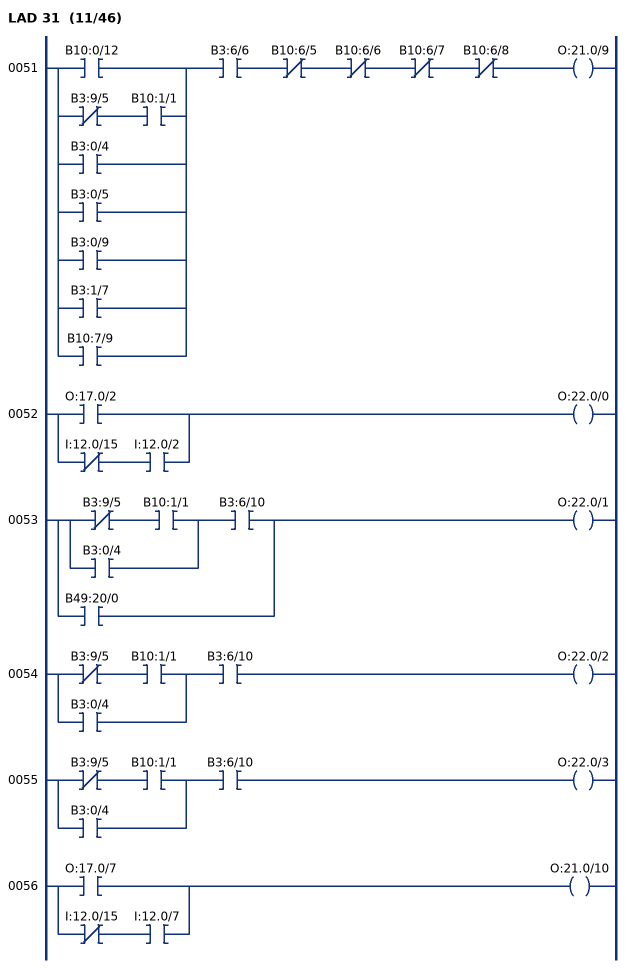
% Rung: 51 %
SOR BST XIC B10:0/12 NXB XIO B3:9/5 XIC B10:1/1 NXB XIC B3:0/4 NXB XIC B3:0/5 NXB XIC B3:0/9 NXB XIC B3:1/7 NXB XIC B10:7/9 BND XIC B3:6/6 XIO B10:6/5 XIO B10:6/6 XIO B10:6/7 XIO B10:6/8 OTE O:21.0/9 EOR
% Rung: 52 %
SOR BST XIC O:17.0/2 NXB XIO I:12.0/15 XIC I:12.0/2 BND OTE O:22.0/0 EOR
% Rung: 53 %
SOR BST BST XIO B3:9/5 XIC B10:1/1 NXB XIC B3:0/4 BND XIC B3:6/10 NXB XIC B49:20/0 BND OTE O:22.0/1 EOR
% Rung: 54 %
SOR BST XIO B3:9/5 XIC B10:1/1 NXB XIC B3:0/4 BND XIC B3:6/10 OTE O:22.0/2 EOR
% Rung: 55 %
SOR BST XIO B3:9/5 XIC B10:1/1 NXB XIC B3:0/4 BND XIC B3:6/10 OTE O:22.0/3 EOR
% Rung: 56 %
SOR BST XIC O:17.0/7 NXB XIO I:12.0/15 XIC I:12.0/7 BND OTE O:21.0/10 EOR

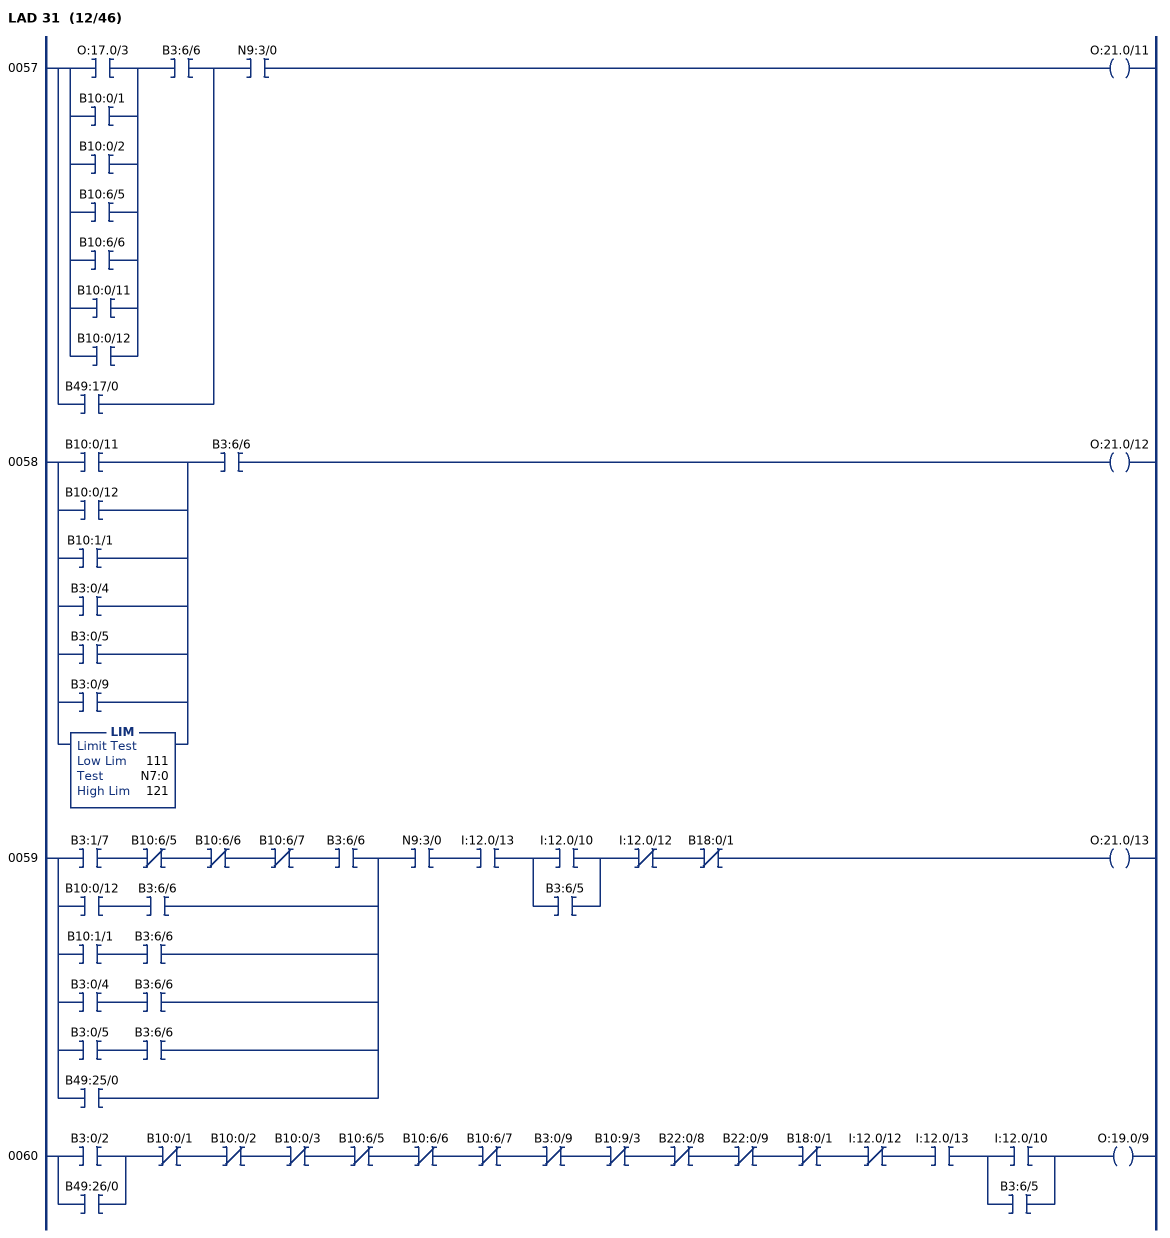
% Rung: 57 %
SOR BST BST XIC O:17.0/3 NXB XIC B10:0/1 NXB XIC B10:0/2 NXB XIC B10:6/5 NXB XIC B10:6/6 NXB XIC B10:0/11 NXB XIC B10:0/12 BND XIC B3:6/6 NXB XIC B49:17/0 BND XIC N9:3/0 OTE O:21.0/11 EOR
% Rung: 58 %
SOR BST XIC B10:0/11 NXB XIC B10:0/12 NXB XIC B10:1/1 NXB XIC B3:0/4 NXB XIC B3:0/5 NXB XIC B3:0/9 NXB LIM 111 N7:0 121 BND XIC B3:6/6 OTE O:21.0/12 EOR
% Rung: 59 %
SOR BST XIC B3:1/7 XIO B10:6/5 XIO B10:6/6 XIO B10:6/7 XIC B3:6/6 NXB XIC B10:0/12 XIC B3:6/6 NXB XIC B10:1/1 XIC B3:6/6 NXB XIC B3:0/4 XIC B3:6/6 NXB XIC B3:0/5 XIC B3:6/6 NXB XIC B49:25/0 BND XIC N9:3/0 XIC I:12.0/13 BST XIC I:12.0/10 NXB XIC B3:6/5 BND XIO I:12.0/12 XIO B18:0/1 OTE O:21.0/13 EOR
% Rung: 60 %
SOR BST XIC B3:0/2 NXB XIC B49:26/0 BND XIO B10:0/1 XIO B10:0/2 XIO B10:0/3 XIO B10:6/5 XIO B10:6/6 XIO B10:6/7 XIO B3:0/9 XIO B10:9/3 XIO B22:0/8 XIO B22:0/9 XIO B18:0/1 XIO I:12.0/12 XIC I:12.0/13 BST XIC I:12.0/10 NXB XIC B3:6/5 BND OTE O:19.0/9 EOR

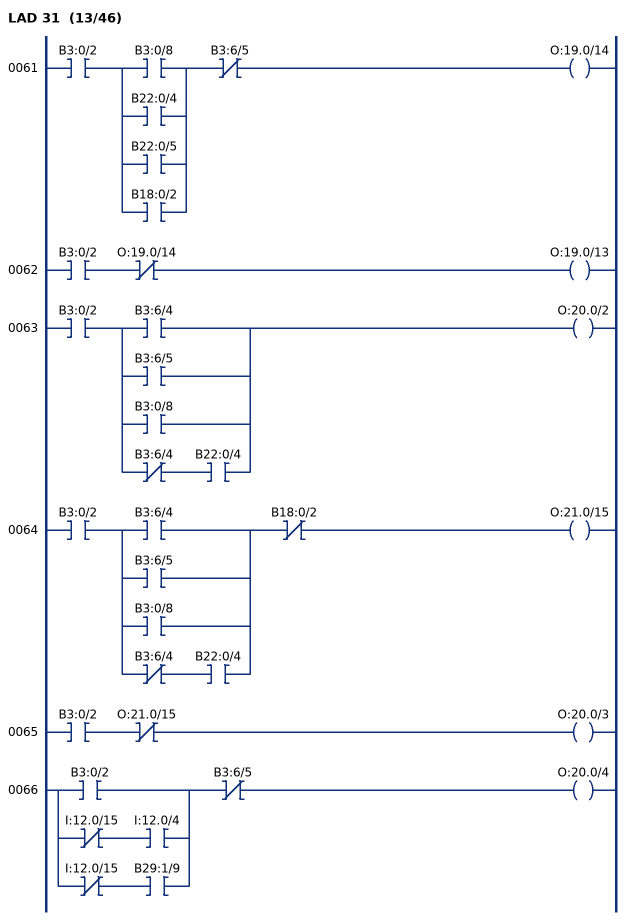
% Rung: 61 %
SOR XIC B3:0/2 BST XIC B3:0/8 NXB XIC B22:0/4 NXB XIC B22:0/5 NXB XIC B18:0/2 BND XIO B3:6/5 OTE O:19.0/14 EOR
% Rung: 62 %
SOR XIC B3:0/2 XIO O:19.0/14 OTE O:19.0/13 EOR
% Rung: 63 %
SOR XIC B3:0/2 BST XIC B3:6/4 NXB XIC B3:6/5 NXB XIC B3:0/8 NXB XIO B3:6/4 XIC B22:0/4 BND OTE O:20.0/2 EOR
% Rung: 64 %
SOR XIC B3:0/2 BST XIC B3:6/4 NXB XIC B3:6/5 NXB XIC B3:0/8 NXB XIO B3:6/4 XIC B22:0/4 BND XIO B18:0/2 OTE O:21.0/15 EOR
% Rung: 65 %
SOR XIC B3:0/2 XIO O:21.0/15 OTE O:20.0/3 EOR
% Rung: 66 %
SOR BST XIC B3:0/2 NXB XIO I:12.0/15 XIC I:12.0/4 NXB XIO I:12.0/15 XIC B29:1/9 BND XIO B3:6/5 OTE O:20.0/4 EOR

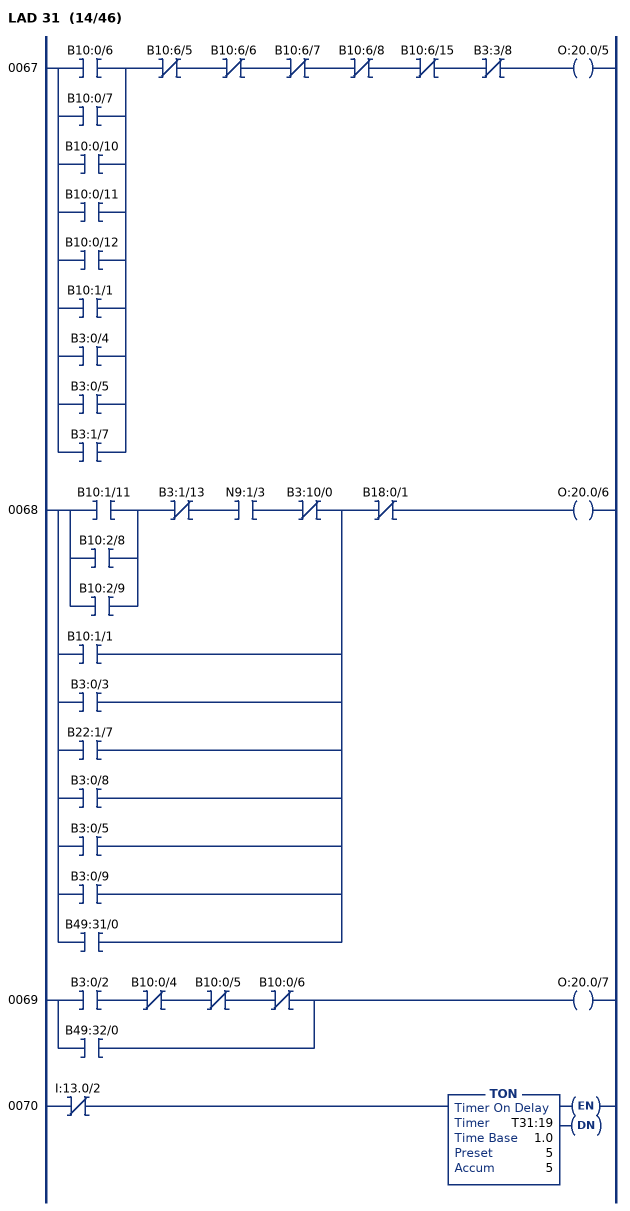
% Rung: 67 %
SOR BST XIC B10:0/6 NXB XIC B10:0/7 NXB XIC B10:0/10 NXB XIC B10:0/11 NXB XIC B10:0/12 NXB XIC B10:1/1 NXB XIC B3:0/4 NXB XIC B3:0/5 NXB XIC B3:1/7 BND XIO B10:6/5 XIO B10:6/6 XIO B10:6/7 XIO B10:6/8 XIO B10:6/15 XIO B3:3/8 OTE O:20.0/5 EOR
% Rung: 68 %
SOR BST BST XIC B10:1/11 NXB XIC B10:2/8 NXB XIC B10:2/9 BND XIO B3:1/13 XIC N9:1/3 XIO B3:10/0 NXB XIC B10:1/1 NXB XIC B3:0/3 NXB XIC B22:1/7 NXB XIC B3:0/8 NXB XIC B3:0/5 NXB XIC B3:0/9 NXB XIC B49:31/0 BND XIO B18:0/1 OTE O:20.0/6 EOR
% Rung: 69 %
SOR BST XIC B3:0/2 XIO B10:0/4 XIO B10:0/5 XIO B10:0/6 NXB XIC B49:32/0 BND OTE O:20.0/7 EOR
% Rung: 70 %
SOR XIO I:13.0/2 TON T31:19 1.0 5 5 EOR

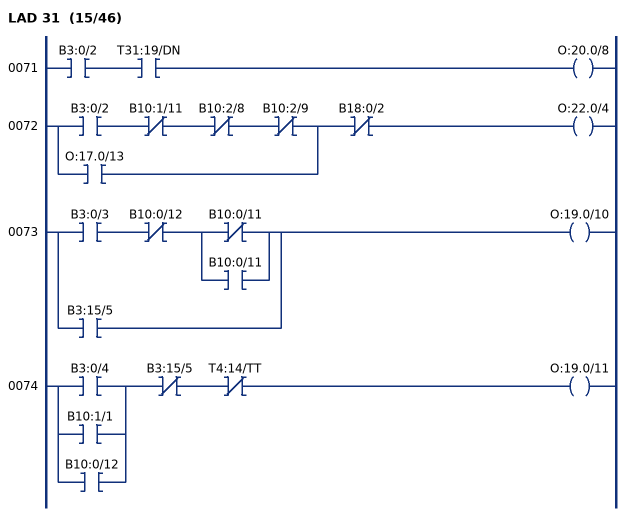
% Rung: 71 %
SOR XIC B3:0/2 XIC T31:19/DN OTE O:20.0/8 EOR
% Rung: 72 %
SOR BST XIC B3:0/2 XIO B10:1/11 XIO B10:2/8 XIO B10:2/9 NXB XIC O:17.0/13 BND XIO B18:0/2 OTE O:22.0/4 EOR
% Rung: 73 %
SOR BST XIC B3:0/3 XIO B10:0/12 BST XIO B10:0/11 NXB XIC B10:0/11 BND NXB XIC B3:15/5 BND OTE O:19.0/10 EOR
% Rung: 74 %
SOR BST XIC B3:0/4 NXB XIC B10:1/1 NXB XIC B10:0/12 BND XIO B3:15/5 XIO T4:14/TT OTE O:19.0/11 EOR

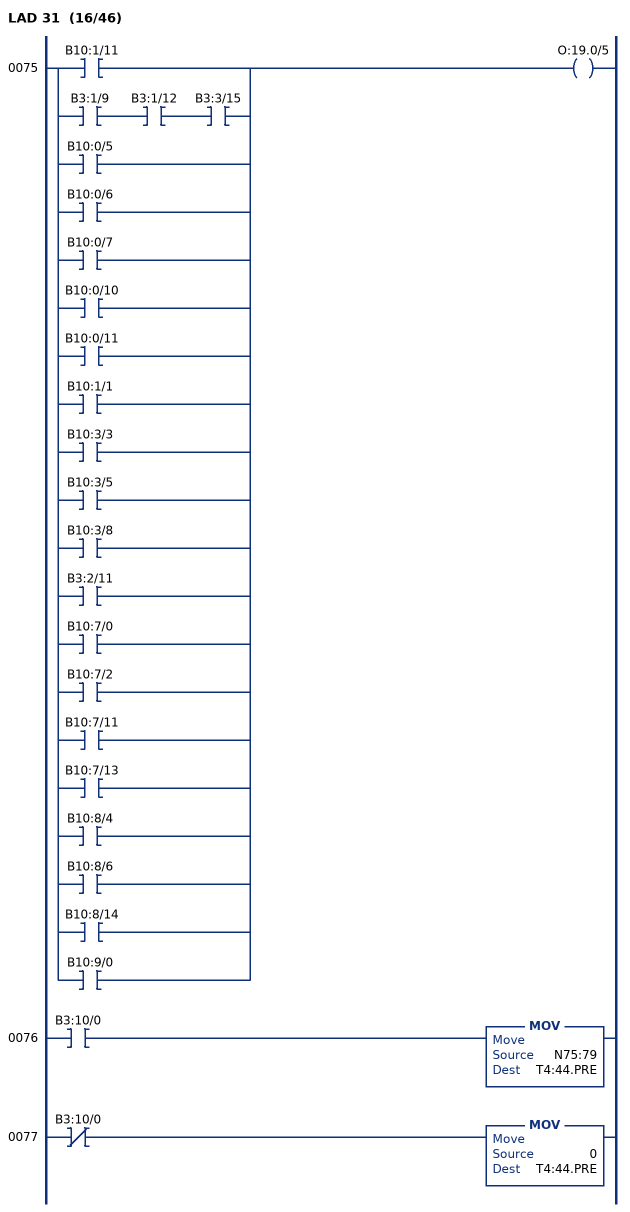
% Rung: 75 %
SOR BST XIC B10:1/11 NXB XIC B3:1/9 XIC B3:1/12 XIC B3:3/15 NXB XIC B10:0/5 NXB XIC B10:0/6 NXB XIC B10:0/7 NXB XIC B10:0/10 NXB XIC B10:0/11 NXB XIC B10:1/1 NXB XIC B10:3/3 NXB XIC B10:3/5 NXB XIC B10:3/8 NXB XIC B3:2/11 NXB XIC B10:7/0 NXB XIC B10:7/2 NXB XIC B10:7/11 NXB XIC B10:7/13 NXB XIC B10:8/4 NXB XIC B10:8/6 NXB XIC B10:8/14 NXB XIC B10:9/0 BND OTE O:19.0/5 EOR
% Rung: 76 %
SOR XIC B3:10/0 MOV N75:79 T4:44.PRE EOR
% Rung: 77 %
SOR XIO B3:10/0 MOV 0 T4:44.PRE EOR

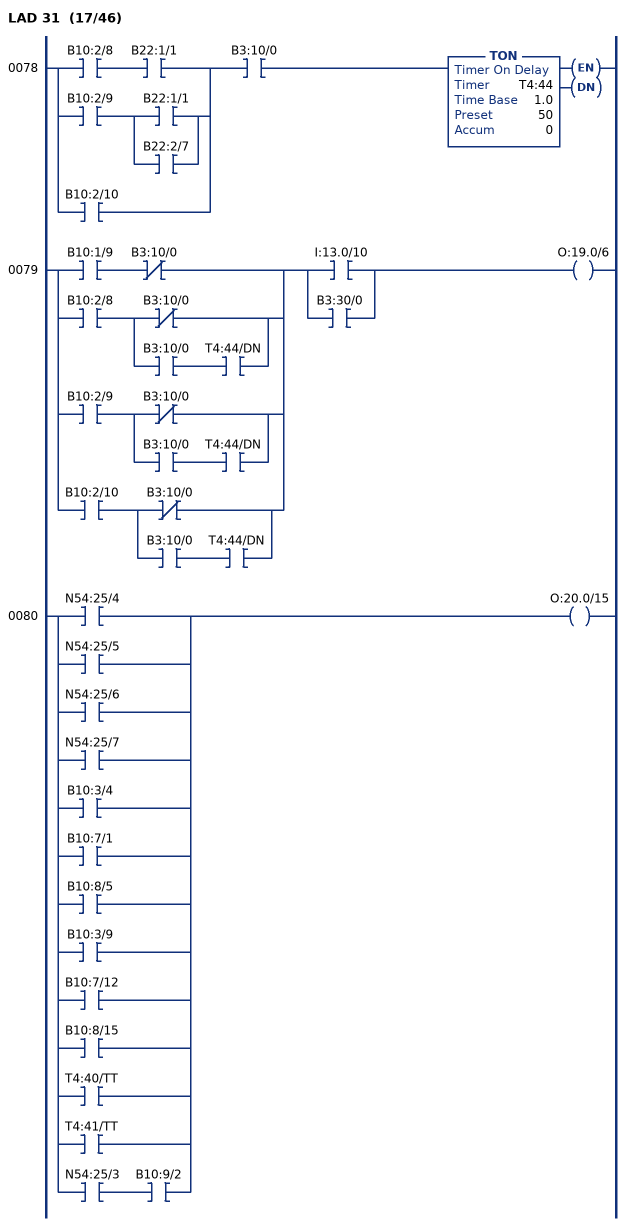
% Rung: 78 %
SOR BST XIC B10:2/8 XIC B22:1/1 NXB XIC B10:2/9 BST XIC B22:1/1 NXB XIC B22:2/7 BND NXB XIC B10:2/10 BND XIC B3:10/0 TON T4:44 1.0 50 0 EOR
% Rung: 79 %
SOR BST XIC B10:1/9 XIO B3:10/0 NXB XIC B10:2/8 BST XIO B3:10/0 NXB XIC B3:10/0 XIC T4:44/DN BND NXB XIC B10:2/9 BST XIO B3:10/0 NXB XIC B3:10/0 XIC T4:44/DN BND NXB XIC B10:2/10 BST XIO B3:10/0 NXB XIC B3:10/0 XIC T4:44/DN BND BND BST XIC I:13.0/10 NXB XIC B3:30/0 BND OTE O:19.0/6 EOR
% Rung: 80 %
SOR BST XIC N54:25/4 NXB XIC N54:25/5 NXB XIC N54:25/6 NXB XIC N54:25/7 NXB XIC B10:3/4 NXB XIC B10:7/1 NXB XIC B10:8/5 NXB XIC B10:3/9 NXB XIC B10:7/12 NXB XIC B10:8/15 NXB XIC T4:40/TT NXB XIC T4:41/TT NXB XIC N54:25/3 XIC B10:9/2 BND OTE O:20.0/15 EOR

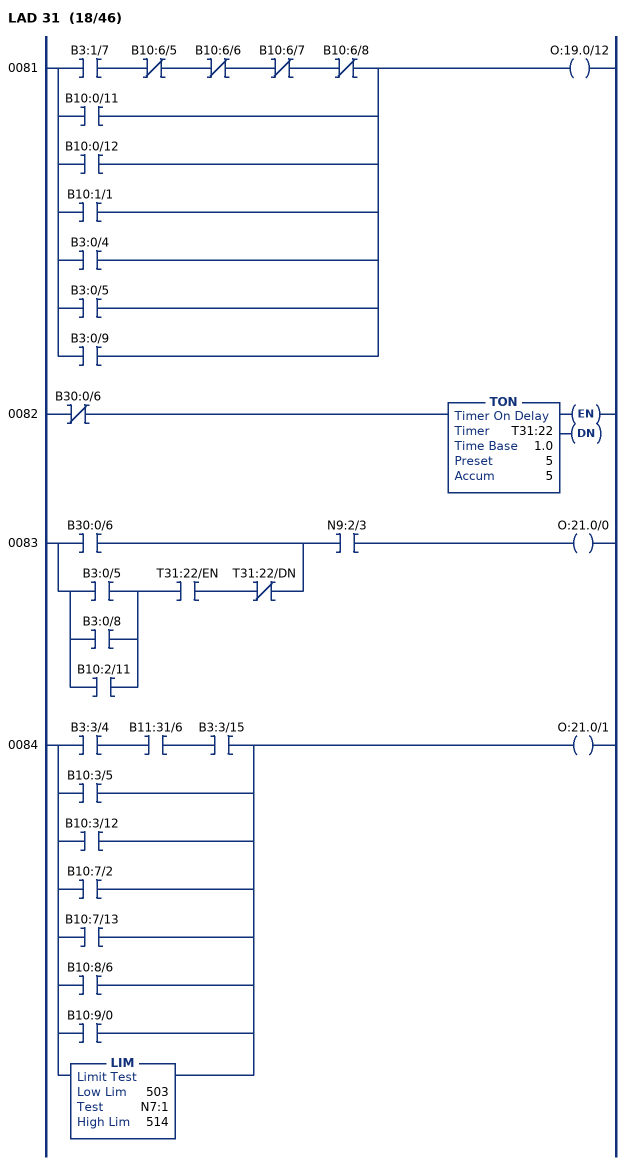
% Rung: 81 %
SOR BST XIC B3:1/7 XIO B10:6/5 XIO B10:6/6 XIO B10:6/7 XIO B10:6/8 NXB XIC B10:0/11 NXB XIC B10:0/12 NXB XIC B10:1/1 NXB XIC B3:0/4 NXB XIC B3:0/5 NXB XIC B3:0/9 BND OTE O:19.0/12 EOR
% Rung: 82 %
SOR XIO B30:0/6 TON T31:22 1.0 5 5 EOR
% Rung: 83 %
SOR BST XIC B30:0/6 NXB BST XIC B3:0/5 NXB XIC B3:0/8 NXB XIC B10:2/11 BND XIC T31:22/EN XIO T31:22/DN BND XIC N9:2/3 OTE O:21.0/0 EOR
% Rung: 84 %
SOR BST XIC B3:3/4 XIC B11:31/6 XIC B3:3/15 NXB BST XIC B10:3/5 NXB XIC B10:3/12 NXB XIC B10:7/2 NXB XIC B10:7/13 NXB XIC B10:8/6 NXB XIC B10:9/0 NXB LIM 503 N7:1 514 BND BND OTE O:21.0/1 EOR

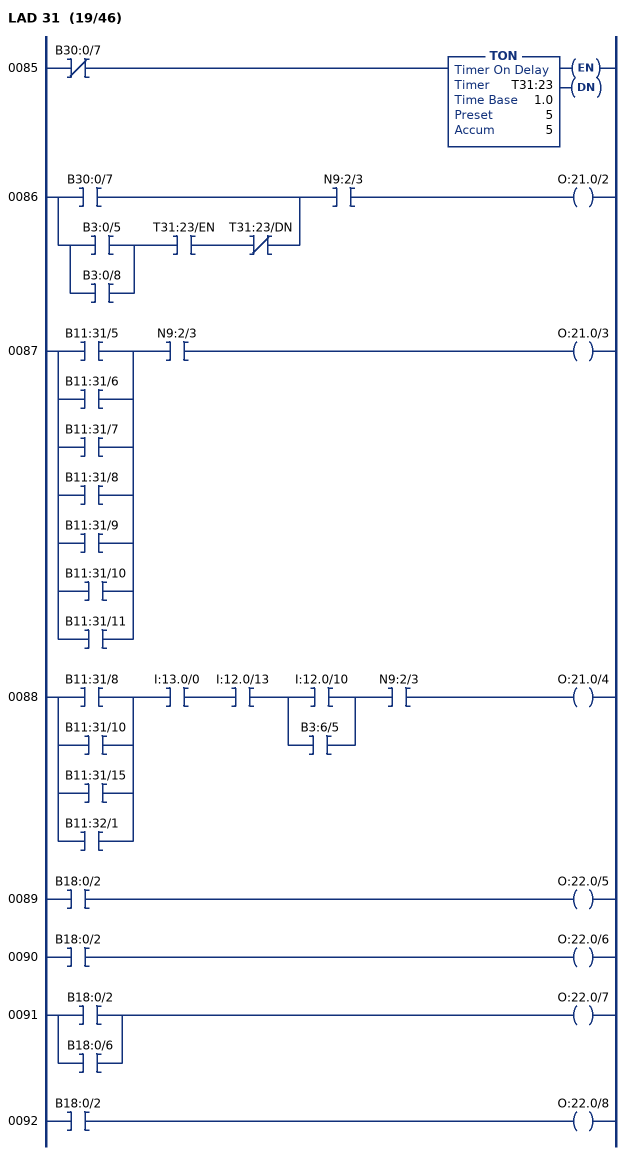
% Rung: 85 %
SOR XIO B30:0/7 TON T31:23 1.0 5 5 EOR
% Rung: 86 %
SOR BST XIC B30:0/7 NXB BST XIC B3:0/5 NXB XIC B3:0/8 BND XIC T31:23/EN XIO T31:23/DN BND XIC N9:2/3 OTE O:21.0/2 EOR
% Rung: 87 %
SOR BST XIC B11:31/5 NXB XIC B11:31/6 NXB XIC B11:31/7 NXB XIC B11:31/8 NXB XIC B11:31/9 NXB XIC B11:31/10 NXB XIC B11:31/11 BND XIC N9:2/3 OTE O:21.0/3 EOR
% Rung: 88 %
SOR BST XIC B11:31/8 NXB XIC B11:31/10 NXB XIC B11:31/15 NXB XIC B11:32/1 BND XIC I:13.0/0 XIC I:12.0/13 BST XIC I:12.0/10 NXB XIC B3:6/5 BND XIC N9:2/3 OTE O:21.0/4 EOR
% Rung: 89 %
SOR XIC B18:0/2 OTE O:22.0/5 EOR
% Rung: 90 %
SOR XIC B18:0/2 OTE O:22.0/6 EOR
% Rung: 91 %
SOR BST XIC B18:0/2 NXB XIC B18:0/6 BND OTE O:22.0/7 EOR
% Rung: 92 %
SOR XIC B18:0/2 OTE O:22.0/8 EOR

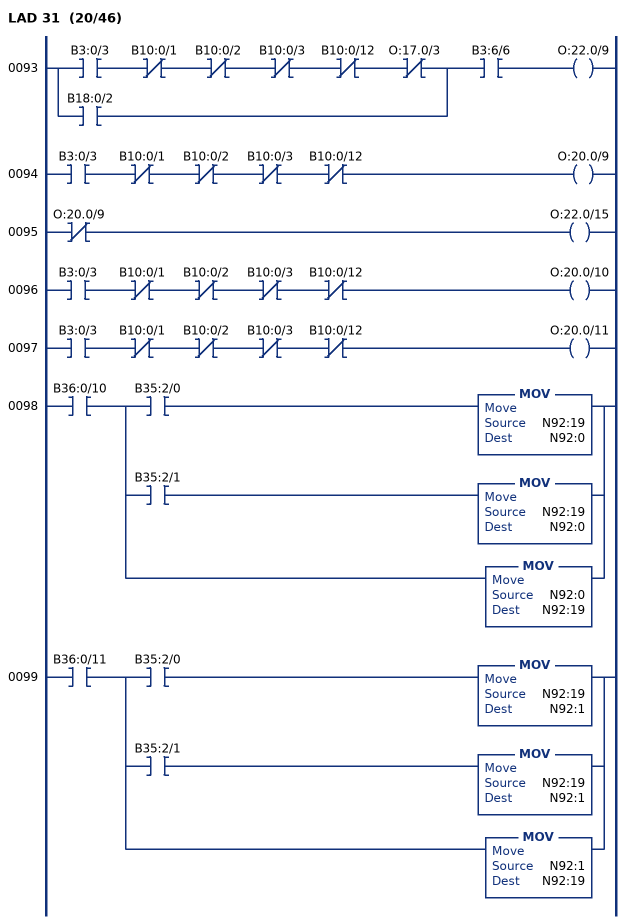
% Rung: 93 %
SOR BST XIC B3:0/3 XIO B10:0/1 XIO B10:0/2 XIO B10:0/3 XIO B10:0/12 XIO O:17.0/3 NXB XIC B18:0/2 BND XIC B3:6/6 OTE O:22.0/9 EOR
% Rung: 94 %
SOR XIC B3:0/3 XIO B10:0/1 XIO B10:0/2 XIO B10:0/3 XIO B10:0/12 OTE O:20.0/9 EOR
% Rung: 95 %
SOR XIO O:20.0/9 OTE O:22.0/15 EOR
% Rung: 96 %
SOR XIC B3:0/3 XIO B10:0/1 XIO B10:0/2 XIO B10:0/3 XIO B10:0/12 OTE O:20.0/10 EOR
% Rung: 97 %
SOR XIC B3:0/3 XIO B10:0/1 XIO B10:0/2 XIO B10:0/3 XIO B10:0/12 OTE O:20.0/11 EOR
% Rung: 98 %
SOR XIC B36:0/10 BST XIC B35:2/0 MOV N92:19 N92:0 NXB XIC B35:2/1 MOV N92:19 N92:0 NXB MOV N92:0 N92:19 BND EOR
% Rung: 99 %
SOR XIC B36:0/11 BST XIC B35:2/0 MOV N92:19 N92:1 NXB XIC B35:2/1 MOV N92:19 N92:1 NXB MOV N92:1 N92:19 BND EOR

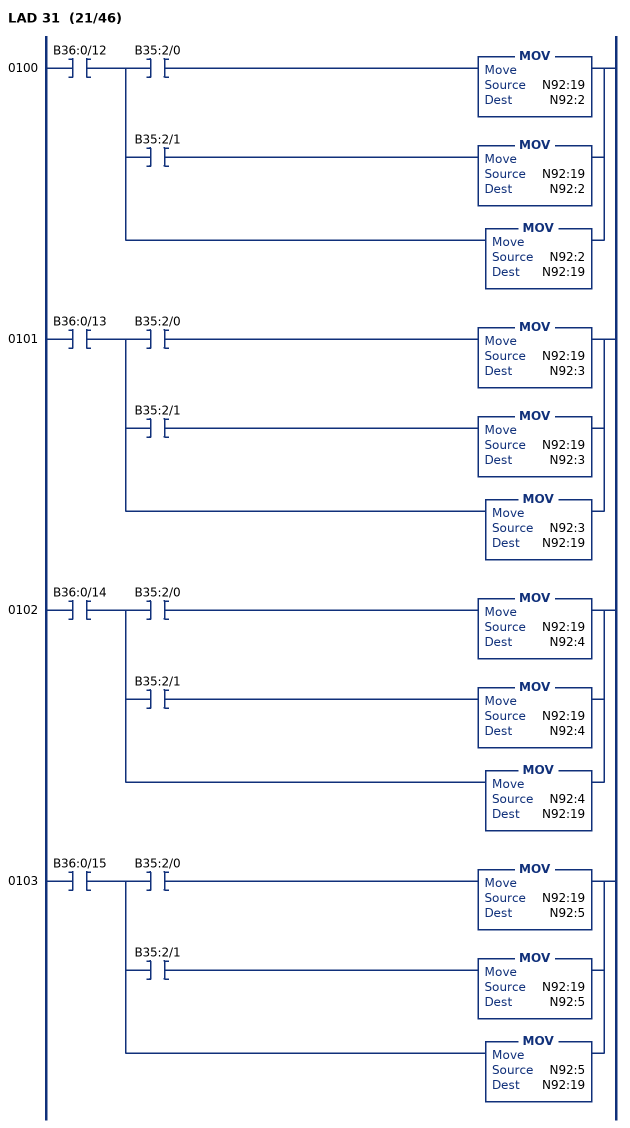
% Rung: 100 %
SOR XIC B36:0/12 BST XIC B35:2/0 MOV N92:19 N92:2 NXB XIC B35:2/1 MOV N92:19 N92:2 NXB MOV N92:2 N92:19 BND EOR
% Rung: 101 %
SOR XIC B36:0/13 BST XIC B35:2/0 MOV N92:19 N92:3 NXB XIC B35:2/1 MOV N92:19 N92:3 NXB MOV N92:3 N92:19 BND EOR
% Rung: 102 %
SOR XIC B36:0/14 BST XIC B35:2/0 MOV N92:19 N92:4 NXB XIC B35:2/1 MOV N92:19 N92:4 NXB MOV N92:4 N92:19 BND EOR
% Rung: 103 %
SOR XIC B36:0/15 BST XIC B35:2/0 MOV N92:19 N92:5 NXB XIC B35:2/1 MOV N92:19 N92:5 NXB MOV N92:5 N92:19 BND EOR

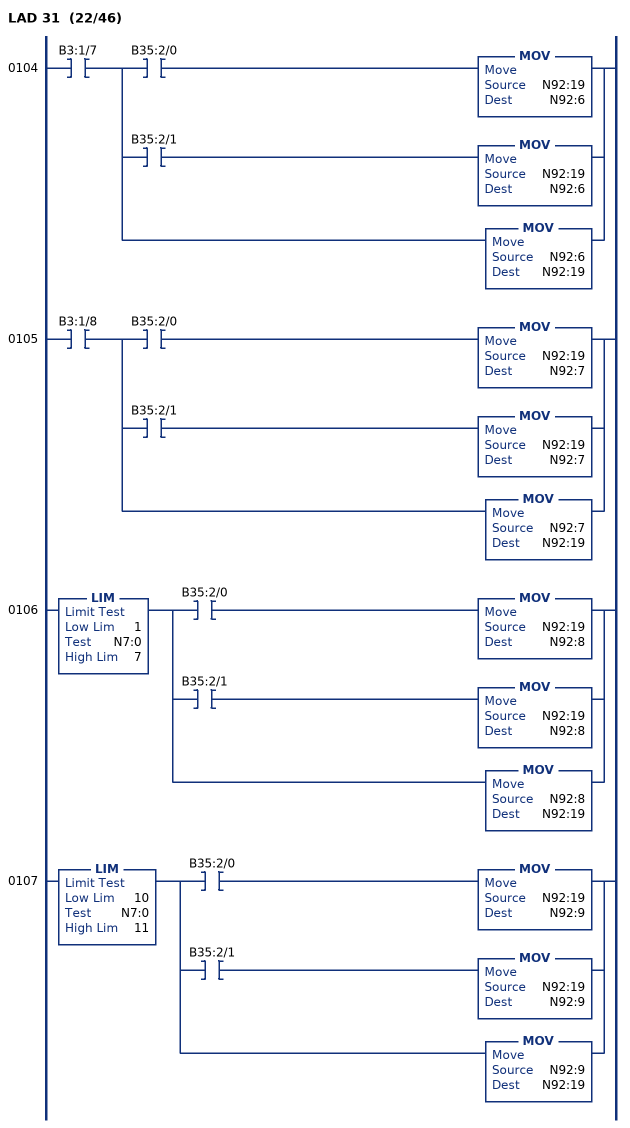
% Rung: 104 %
SOR XIC B3:1/7 BST XIC B35:2/0 MOV N92:19 N92:6 NXB XIC B35:2/1 MOV N92:19 N92:6 NXB MOV N92:6 N92:19 BND EOR
% Rung: 105 %
SOR XIC B3:1/8 BST XIC B35:2/0 MOV N92:19 N92:7 NXB XIC B35:2/1 MOV N92:19 N92:7 NXB MOV N92:7 N92:19 BND EOR
% Rung: 106 %
SOR LIM 1 N7:0 7 BST XIC B35:2/0 MOV N92:19 N92:8 NXB XIC B35:2/1 MOV N92:19 N92:8 NXB MOV N92:8 N92:19 BND EOR
% Rung: 107 %
SOR LIM 10 N7:0 11 BST XIC B35:2/0 MOV N92:19 N92:9 NXB XIC B35:2/1 MOV N92:19 N92:9 NXB MOV N92:9 N92:19 BND EOR

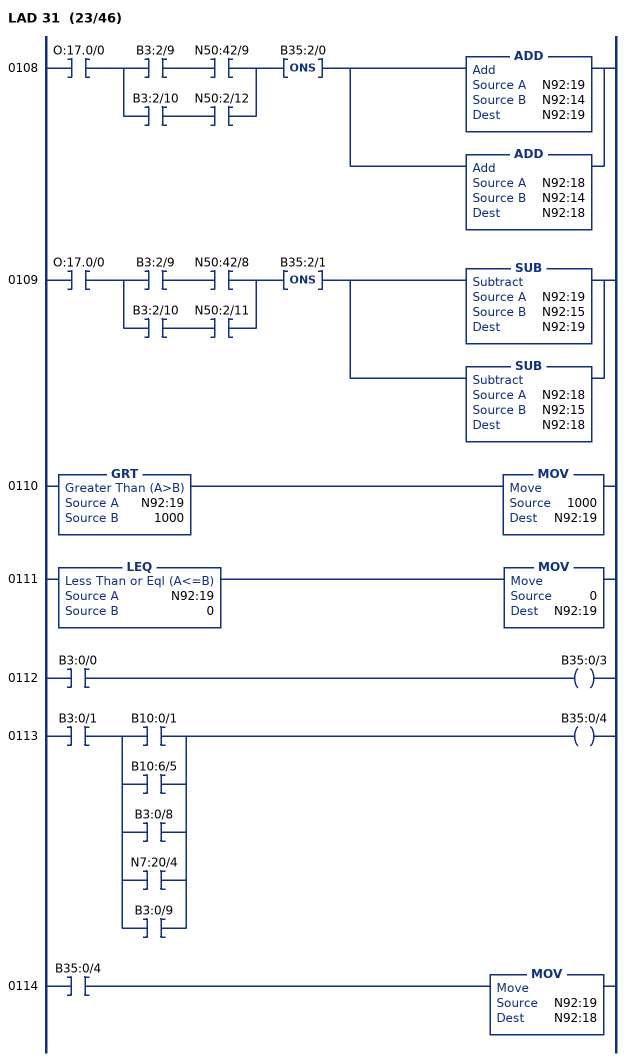
% Rung: 108 %
SOR XIC O:17.0/0 BST XIC B3:2/9 XIC N50:42/9 NXB XIC B3:2/10 XIC N50:2/12 BND OSR B35:2/0 BST ADD N92:19 N92:14 N92:19 NXB ADD N92:18 N92:14 N92:18 BND EOR
% Rung: 109 %
SOR XIC O:17.0/0 BST XIC B3:2/9 XIC N50:42/8 NXB XIC B3:2/10 XIC N50:2/11 BND OSR B35:2/1 BST SUB N92:19 N92:15 N92:19 NXB SUB N92:18 N92:15 N92:18 BND EOR
% Rung: 110 %
SOR GRT N92:19 1000 MOV 1000 N92:19 EOR
% Rung: 111 %
SOR LEQ N92:19 0 MOV 0 N92:19 EOR
% Rung: 112 %
SOR XIC B3:0/0 OTE B35:0/3 EOR
% Rung: 113 %
SOR XIC B3:0/1 BST XIC B10:0/1 NXB XIC B10:6/5 NXB XIC B3:0/8 NXB XIC N7:20/4 NXB XIC B3:0/9 BND OTE B35:0/4 EOR
% Rung: 114 %
SOR XIC B35:0/4 MOV N92:19 N92:18 EOR

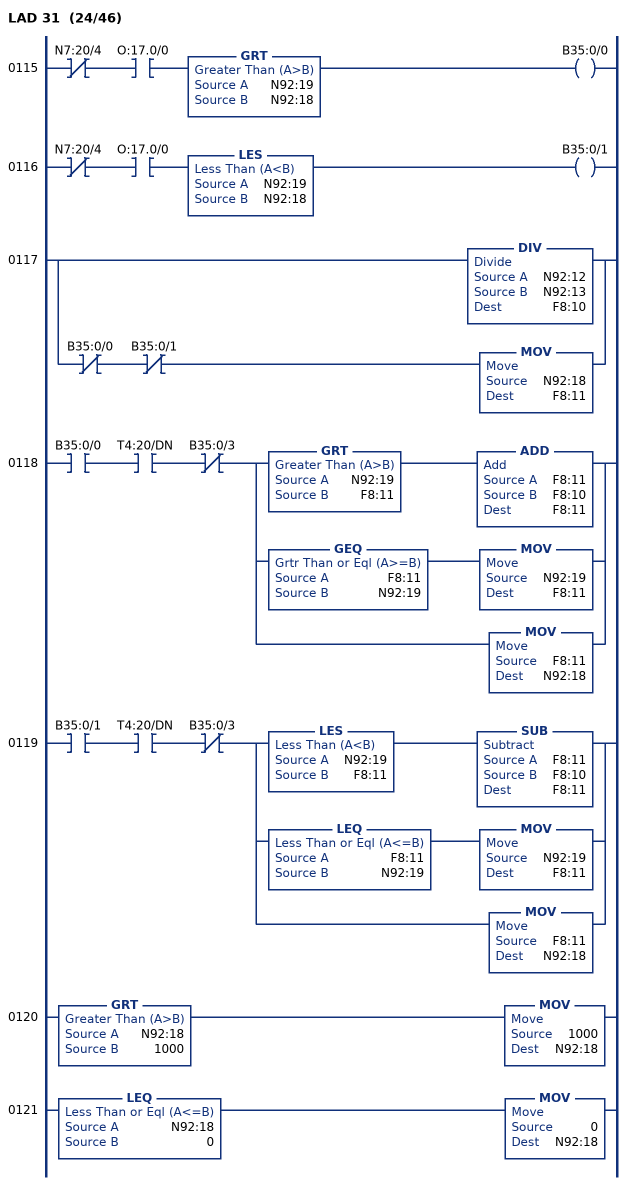
% Rung: 115 %
SOR XIO N7:20/4 XIC O:17.0/0 GRT N92:19 N92:18 OTE B35:0/0 EOR
% Rung: 116 %
SOR XIO N7:20/4 XIC O:17.0/0 LES N92:19 N92:18 OTE B35:0/1 EOR
% Rung: 117 %
SOR BST DIV N92:12 N92:13 F8:10 NXB XIO B35:0/0 XIO B35:0/1 MOV N92:18 F8:11 BND EOR
% Rung: 118 %
SOR XIC B35:0/0 XIC T4:20/DN XIO B35:0/3 BST GRT N92:19 F8:11 ADD F8:11 F8:10 F8:11 NXB GEQ F8:11 N92:19 MOV N92:19 F8:11 NXB MOV F8:11 N92:18 BND EOR
% Rung: 119 %
SOR XIC B35:0/1 XIC T4:20/DN XIO B35:0/3 BST LES N92:19 F8:11 SUB F8:11 F8:10 F8:11 NXB LEQ F8:11 N92:19 MOV N92:19 F8:11 NXB MOV F8:11 N92:18 BND EOR
% Rung: 120 %
SOR GRT N92:18 1000 MOV 1000 N92:18 EOR
% Rung: 121 %
SOR LEQ N92:18 0 MOV 0 N92:18 EOR

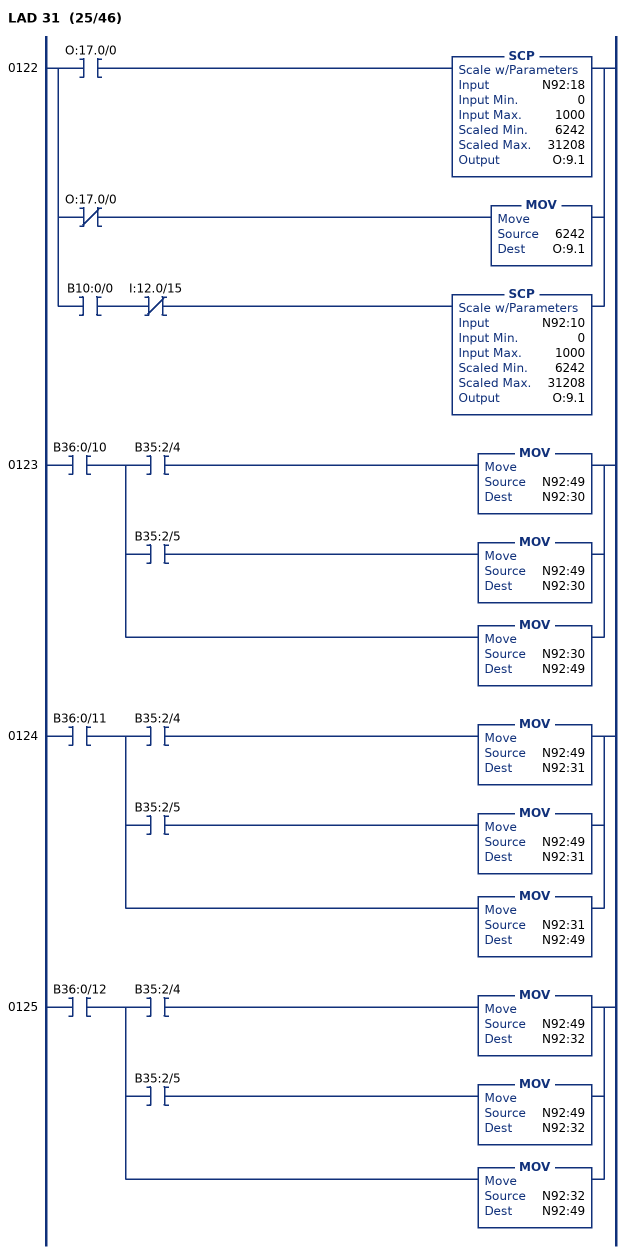
% Rung: 122 %
SOR BST XIC O:17.0/0 SCP N92:18 0 1000 6242 31208 O:9.1 NXB XIO O:17.0/0 MOV 6242 O:9.1 NXB XIC B10:0/0 XIO I:12.0/15 SCP N92:10 0 1000 6242 31208 O:9.1 BND EOR
% Rung: 123 %
SOR XIC B36:0/10 BST XIC B35:2/4 MOV N92:49 N92:30 NXB XIC B35:2/5 MOV N92:49 N92:30 NXB MOV N92:30 N92:49 BND EOR
% Rung: 124 %
SOR XIC B36:0/11 BST XIC B35:2/4 MOV N92:49 N92:31 NXB XIC B35:2/5 MOV N92:49 N92:31 NXB MOV N92:31 N92:49 BND EOR
% Rung: 125 %
SOR XIC B36:0/12 BST XIC B35:2/4 MOV N92:49 N92:32 NXB XIC B35:2/5 MOV N92:49 N92:32 NXB MOV N92:32 N92:49 BND EOR

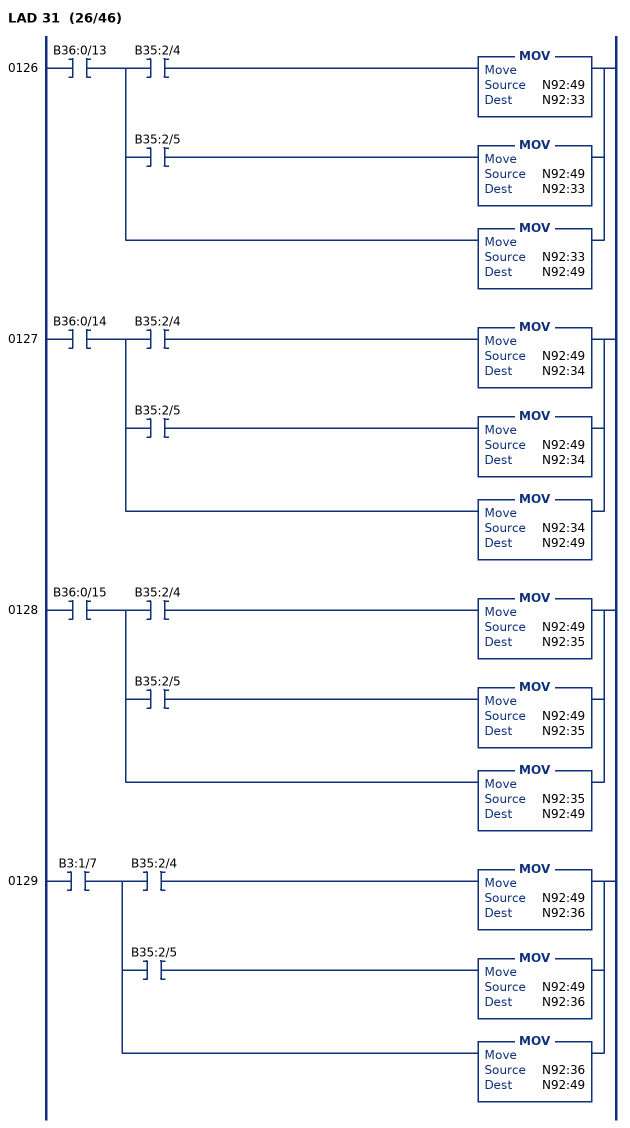
% Rung: 126 %
SOR XIC B36:0/13 BST XIC B35:2/4 MOV N92:49 N92:33 NXB XIC B35:2/5 MOV N92:49 N92:33 NXB MOV N92:33 N92:49 BND EOR
% Rung: 127 %
SOR XIC B36:0/14 BST XIC B35:2/4 MOV N92:49 N92:34 NXB XIC B35:2/5 MOV N92:49 N92:34 NXB MOV N92:34 N92:49 BND EOR
% Rung: 128 %
SOR XIC B36:0/15 BST XIC B35:2/4 MOV N92:49 N92:35 NXB XIC B35:2/5 MOV N92:49 N92:35 NXB MOV N92:35 N92:49 BND EOR
% Rung: 129 %
SOR XIC B3:1/7 BST XIC B35:2/4 MOV N92:49 N92:36 NXB XIC B35:2/5 MOV N92:49 N92:36 NXB MOV N92:36 N92:49 BND EOR

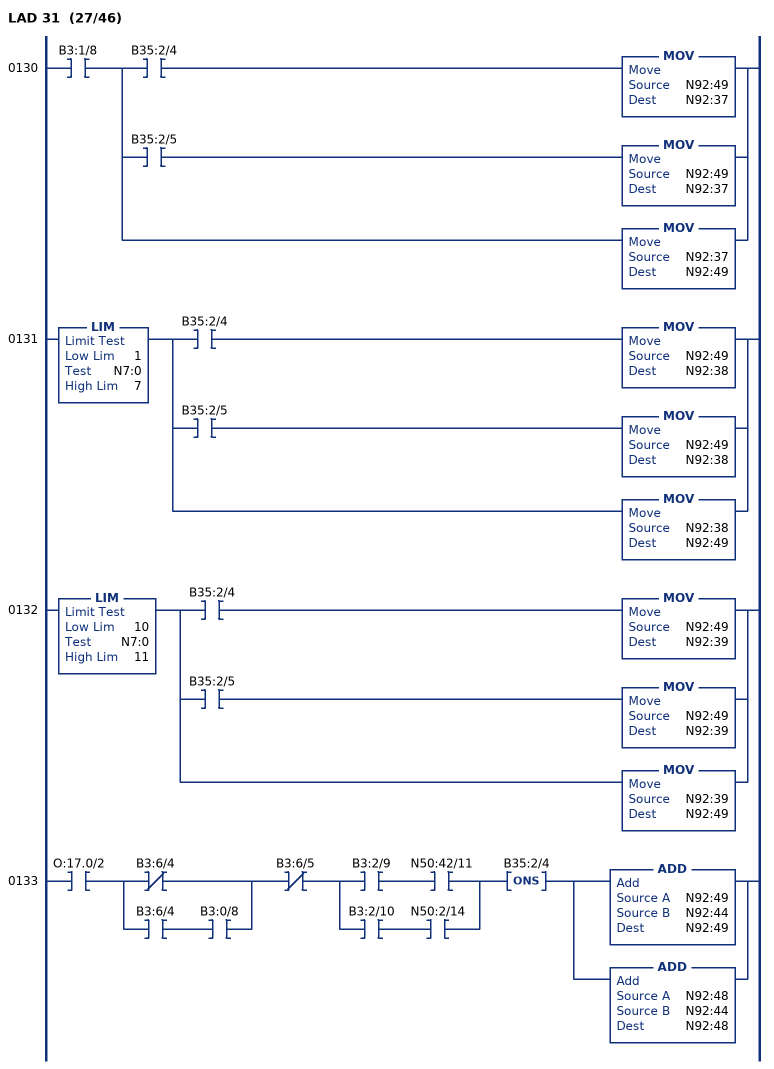
% Rung: 130 %
SOR XIC B3:1/8 BST XIC B35:2/4 MOV N92:49 N92:37 NXB XIC B35:2/5 MOV N92:49 N92:37 NXB MOV N92:37 N92:49 BND EOR
% Rung: 131 %
SOR LIM 1 N7:0 7 BST XIC B35:2/4 MOV N92:49 N92:38 NXB XIC B35:2/5 MOV N92:49 N92:38 NXB MOV N92:38 N92:49 BND EOR
% Rung: 132 %
SOR LIM 10 N7:0 11 BST XIC B35:2/4 MOV N92:49 N92:39 NXB XIC B35:2/5 MOV N92:49 N92:39 NXB MOV N92:39 N92:49 BND EOR
% Rung: 133 %
SOR XIC O:17.0/2 BST XIO B3:6/4 NXB XIC B3:6/4 XIC B3:0/8 BND XIO B3:6/5 BST XIC B3:2/9 XIC N50:42/11 NXB XIC B3:2/10 XIC N50:2/14 BND OSR B35:2/4 BST ADD N92:49 N92:44 N92:49 NXB ADD N92:48 N92:44 N92:48 BND EOR

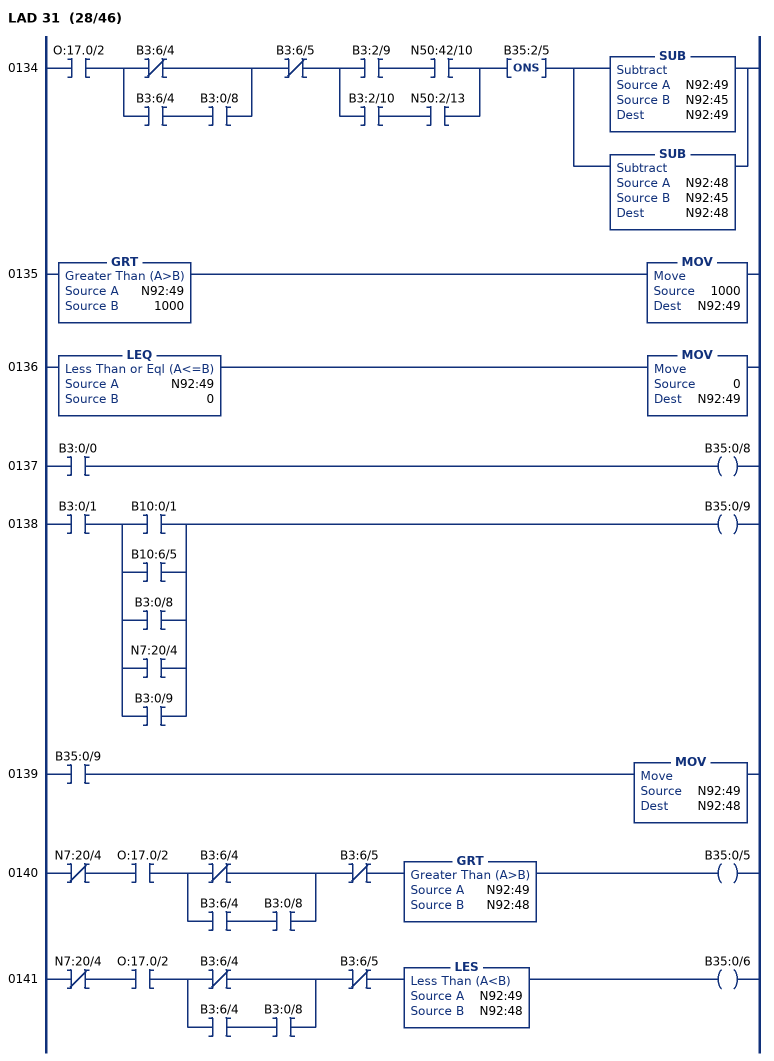
% Rung: 134 %
SOR XIC O:17.0/2 BST XIO B3:6/4 NXB XIC B3:6/4 XIC B3:0/8 BND XIO B3:6/5 BST XIC B3:2/9 XIC N50:42/10 NXB XIC B3:2/10 XIC N50:2/13 BND OSR B35:2/5 BST SUB N92:49 N92:45 N92:49 NXB SUB N92:48 N92:45 N92:48 BND EOR
% Rung: 135 %
SOR GRT N92:49 1000 MOV 1000 N92:49 EOR
% Rung: 136 %
SOR LEQ N92:49 0 MOV 0 N92:49 EOR
% Rung: 137 %
SOR XIC B3:0/0 OTE B35:0/8 EOR
% Rung: 138 %
SOR XIC B3:0/1 BST XIC B10:0/1 NXB XIC B10:6/5 NXB XIC B3:0/8 NXB XIC N7:20/4 NXB XIC B3:0/9 BND OTE B35:0/9 EOR
% Rung: 139 %
SOR XIC B35:0/9 MOV N92:49 N92:48 EOR
% Rung: 140 %
SOR XIO N7:20/4 XIC O:17.0/2 BST XIO B3:6/4 NXB XIC B3:6/4 XIC B3:0/8 BND XIO B3:6/5 GRT N92:49 N92:48 OTE B35:0/5 EOR
% Rung: 141 %
SOR XIO N7:20/4 XIC O:17.0/2 BST XIO B3:6/4 NXB XIC B3:6/4 XIC B3:0/8 BND XIO B3:6/5 LES N92:49 N92:48 OTE B35:0/6 EOR

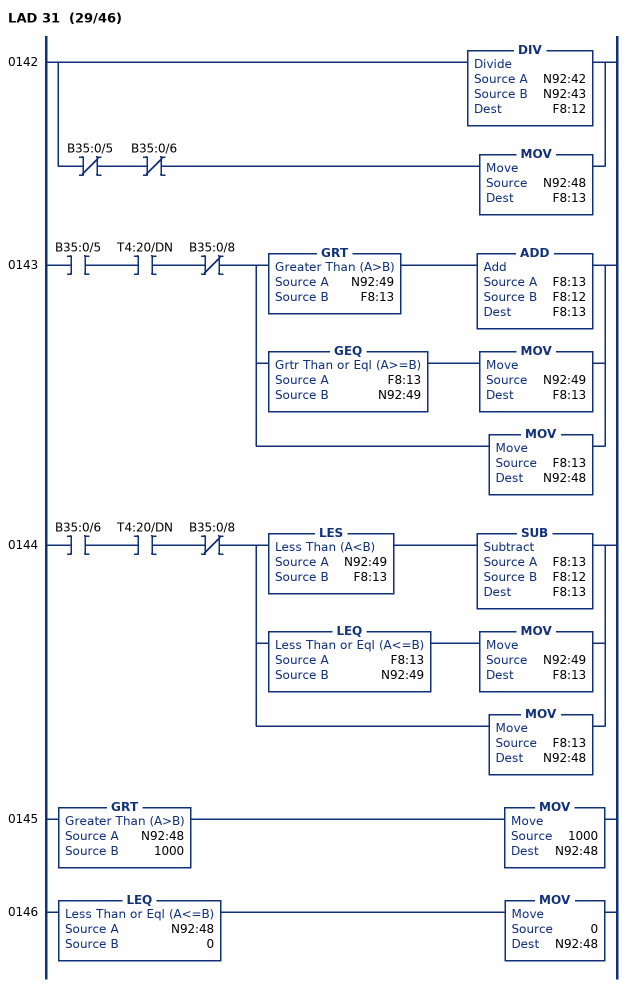
% Rung: 142 %
SOR BST DIV N92:42 N92:43 F8:12 NXB XIO B35:0/5 XIO B35:0/6 MOV N92:48 F8:13 BND EOR
% Rung: 143 %
SOR XIC B35:0/5 XIC T4:20/DN XIO B35:0/8 BST GRT N92:49 F8:13 ADD F8:13 F8:12 F8:13 NXB GEQ F8:13 N92:49 MOV N92:49 F8:13 NXB MOV F8:13 N92:48 BND EOR
% Rung: 144 %
SOR XIC B35:0/6 XIC T4:20/DN XIO B35:0/8 BST LES N92:49 F8:13 SUB F8:13 F8:12 F8:13 NXB LEQ F8:13 N92:49 MOV N92:49 F8:13 NXB MOV F8:13 N92:48 BND EOR
% Rung: 145 %
SOR GRT N92:48 1000 MOV 1000 N92:48 EOR
% Rung: 146 %
SOR LEQ N92:48 0 MOV 0 N92:48 EOR

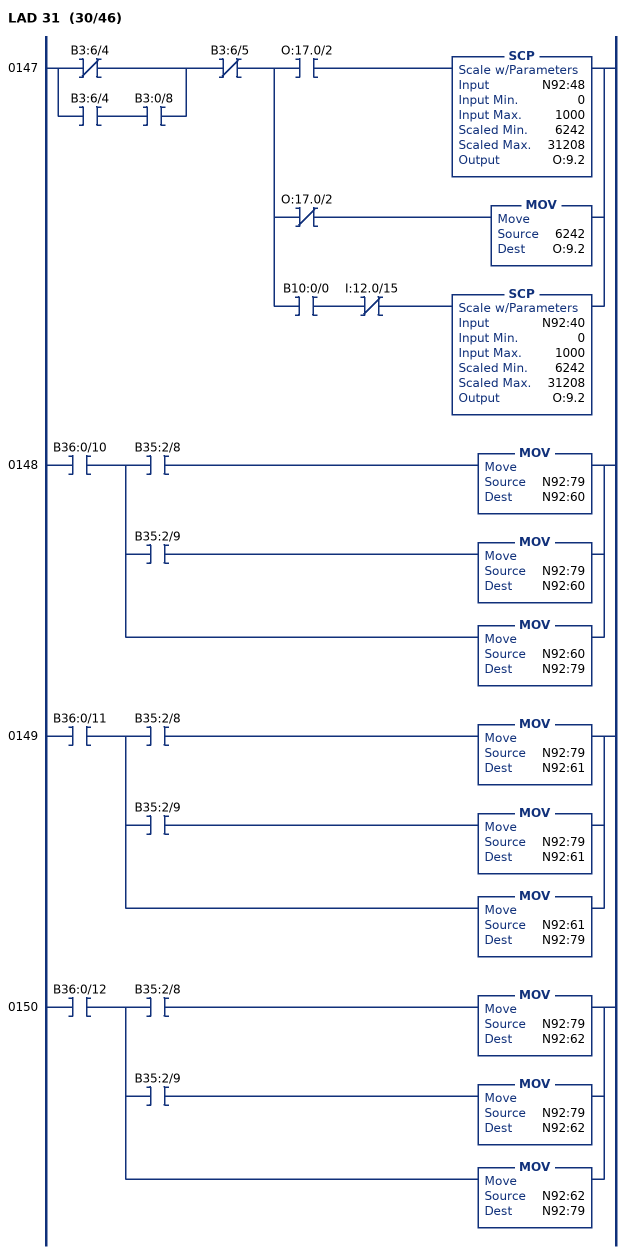
% Rung: 147 %
SOR BST XIO B3:6/4 NXB XIC B3:6/4 XIC B3:0/8 BND XIO B3:6/5 BST XIC O:17.0/2 SCP N92:48 0 1000 6242 31208 O:9.2 NXB XIO O:17.0/2 MOV 6242 O:9.2 NXB XIC B10:0/0 XIO I:12.0/15 SCP N92:40 0 1000 6242 31208 O:9.2 BND EOR
% Rung: 148 %
SOR XIC B36:0/10 BST XIC B35:2/8 MOV N92:79 N92:60 NXB XIC B35:2/9 MOV N92:79 N92:60 NXB MOV N92:60 N92:79 BND EOR
% Rung: 149 %
SOR XIC B36:0/11 BST XIC B35:2/8 MOV N92:79 N92:61 NXB XIC B35:2/9 MOV N92:79 N92:61 NXB MOV N92:61 N92:79 BND EOR
% Rung: 150 %
SOR XIC B36:0/12 BST XIC B35:2/8 MOV N92:79 N92:62 NXB XIC B35:2/9 MOV N92:79 N92:62 NXB MOV N92:62 N92:79 BND EOR

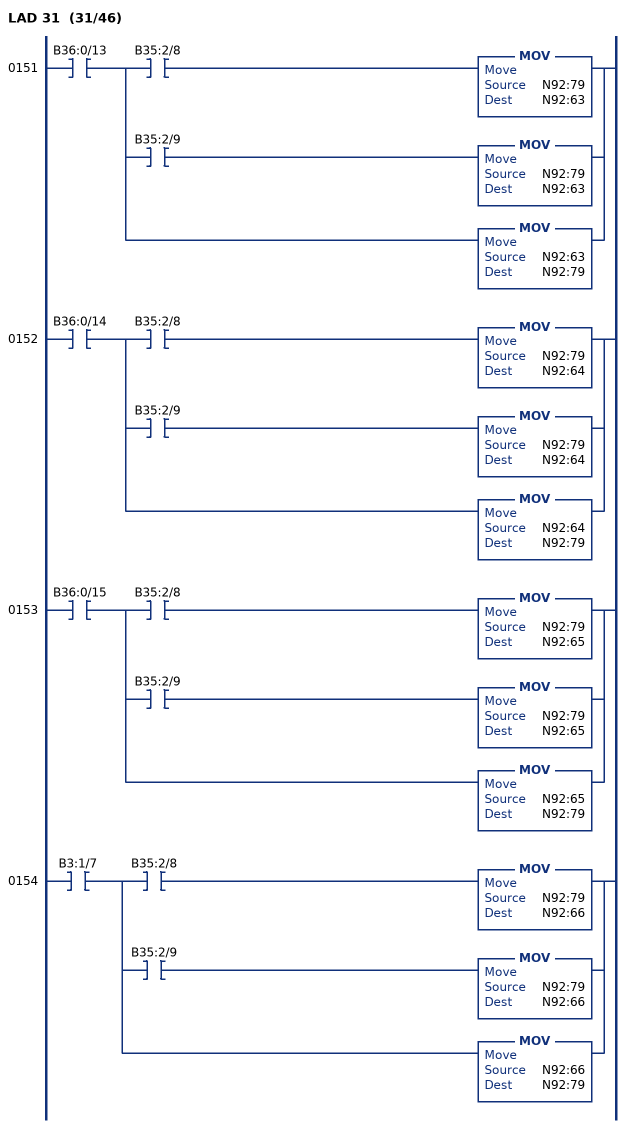
% Rung: 151 %
SOR XIC B36:0/13 BST XIC B35:2/8 MOV N92:79 N92:63 NXB XIC B35:2/9 MOV N92:79 N92:63 NXB MOV N92:63 N92:79 BND EOR
% Rung: 152 %
SOR XIC B36:0/14 BST XIC B35:2/8 MOV N92:79 N92:64 NXB XIC B35:2/9 MOV N92:79 N92:64 NXB MOV N92:64 N92:79 BND EOR
% Rung: 153 %
SOR XIC B36:0/15 BST XIC B35:2/8 MOV N92:79 N92:65 NXB XIC B35:2/9 MOV N92:79 N92:65 NXB MOV N92:65 N92:79 BND EOR
% Rung: 154 %
SOR XIC B3:1/7 BST XIC B35:2/8 MOV N92:79 N92:66 NXB XIC B35:2/9 MOV N92:79 N92:66 NXB MOV N92:66 N92:79 BND EOR

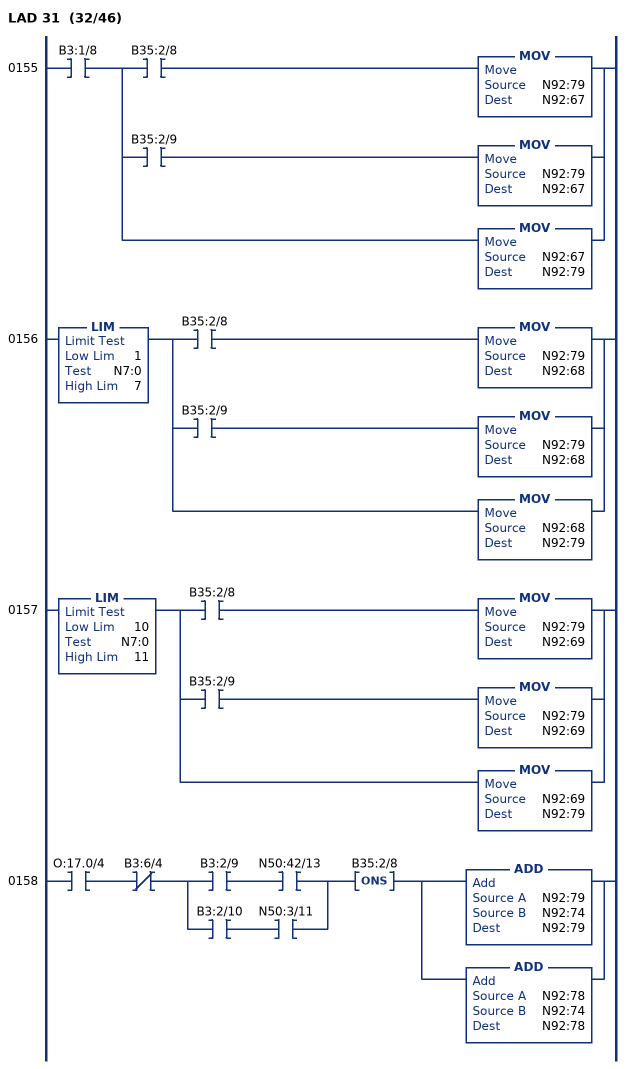
% Rung: 155 %
SOR XIC B3:1/8 BST XIC B35:2/8 MOV N92:79 N92:67 NXB XIC B35:2/9 MOV N92:79 N92:67 NXB MOV N92:67 N92:79 BND EOR
% Rung: 156 %
SOR LIM 1 N7:0 7 BST XIC B35:2/8 MOV N92:79 N92:68 NXB XIC B35:2/9 MOV N92:79 N92:68 NXB MOV N92:68 N92:79 BND EOR
% Rung: 157 %
SOR LIM 10 N7:0 11 BST XIC B35:2/8 MOV N92:79 N92:69 NXB XIC B35:2/9 MOV N92:79 N92:69 NXB MOV N92:69 N92:79 BND EOR
% Rung: 158 %
SOR XIC O:17.0/4 XIO B3:6/4 BST XIC B3:2/9 XIC N50:42/13 NXB XIC B3:2/10 XIC N50:3/11 BND OSR B35:2/8 BST ADD N92:79 N92:74 N92:79 NXB ADD N92:78 N92:74 N92:78 BND EOR

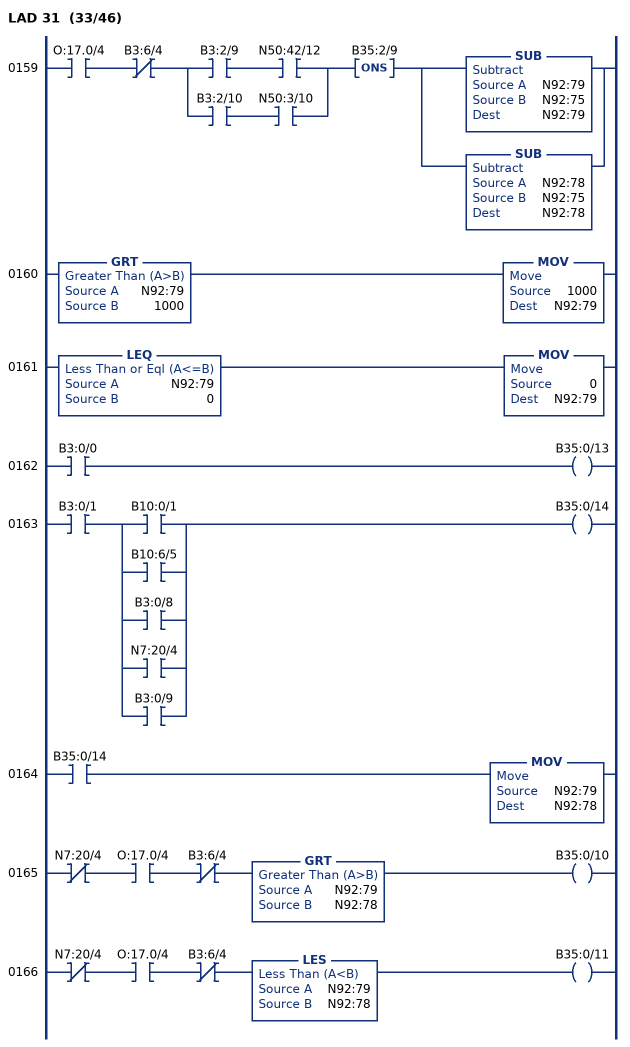
% Rung: 159 %
SOR XIC O:17.0/4 XIO B3:6/4 BST XIC B3:2/9 XIC N50:42/12 NXB XIC B3:2/10 XIC N50:3/10 BND OSR B35:2/9 BST SUB N92:79 N92:75 N92:79 NXB SUB N92:78 N92:75 N92:78 BND EOR
% Rung: 160 %
SOR GRT N92:79 1000 MOV 1000 N92:79 EOR
% Rung: 161 %
SOR LEQ N92:79 0 MOV 0 N92:79 EOR
% Rung: 162 %
SOR XIC B3:0/0 OTE B35:0/13 EOR
% Rung: 163 %
SOR XIC B3:0/1 BST XIC B10:0/1 NXB XIC B10:6/5 NXB XIC B3:0/8 NXB XIC N7:20/4 NXB XIC B3:0/9 BND OTE B35:0/14 EOR
% Rung: 164 %
SOR XIC B35:0/14 MOV N92:79 N92:78 EOR
% Rung: 165 %
SOR XIO N7:20/4 XIC O:17.0/4 XIO B3:6/4 GRT N92:79 N92:78 OTE B35:0/10 EOR
% Rung: 166 %
SOR XIO N7:20/4 XIC O:17.0/4 XIO B3:6/4 LES N92:79 N92:78 OTE B35:0/11 EOR

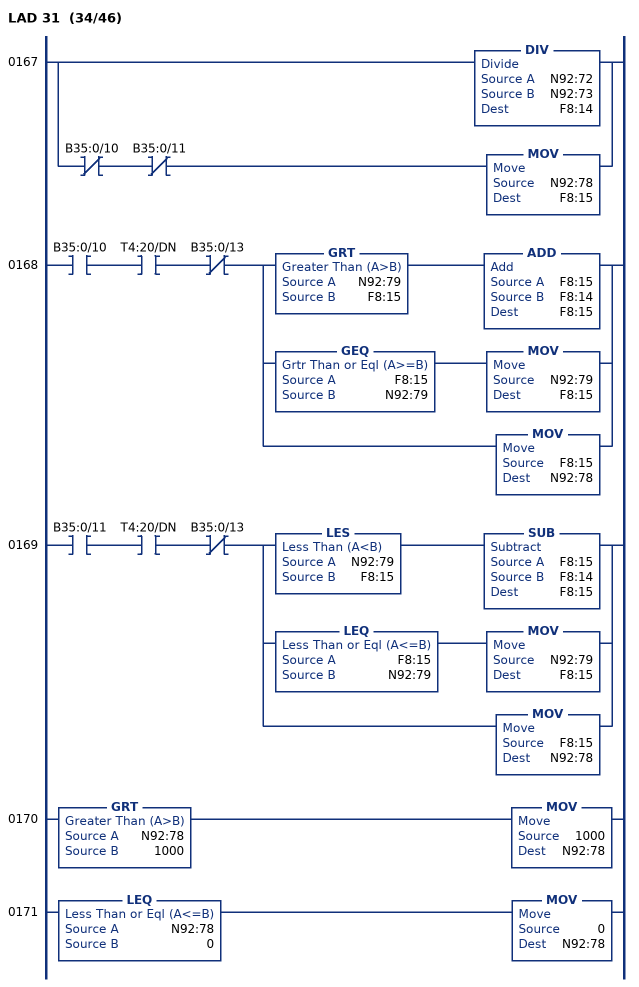
% Rung: 167 %
SOR BST DIV N92:72 N92:73 F8:14 NXB XIO B35:0/10 XIO B35:0/11 MOV N92:78 F8:15 BND EOR
% Rung: 168 %
SOR XIC B35:0/10 XIC T4:20/DN XIO B35:0/13 BST GRT N92:79 F8:15 ADD F8:15 F8:14 F8:15 NXB GEQ F8:15 N92:79 MOV N92:79 F8:15 NXB MOV F8:15 N92:78 BND EOR
% Rung: 169 %
SOR XIC B35:0/11 XIC T4:20/DN XIO B35:0/13 BST LES N92:79 F8:15 SUB F8:15 F8:14 F8:15 NXB LEQ F8:15 N92:79 MOV N92:79 F8:15 NXB MOV F8:15 N92:78 BND EOR
% Rung: 170 %
SOR GRT N92:78 1000 MOV 1000 N92:78 EOR
% Rung: 171 %
SOR LEQ N92:78 0 MOV 0 N92:78 EOR

